// Mitsubishi GX Works2 project: Jesús Beato 2023-1283 #3   PLC: Q00J

PROGRAM MAIN
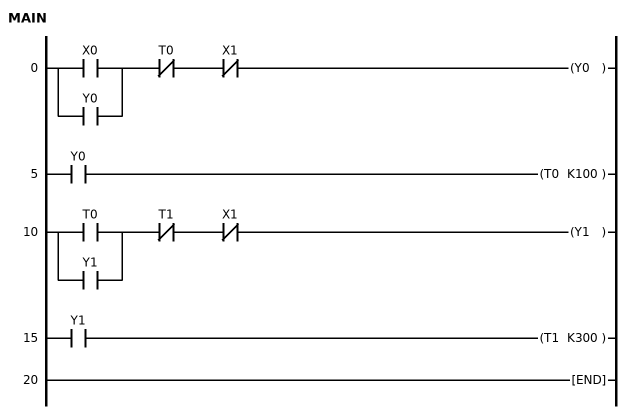
0     LD      X0
      OR      Y0
      ANI     T0
      ANI     X1
      OUT     Y0
5     LD      Y0
      OUT     T0 K100
10    LD      T0
      OR      Y1
      ANI     T1
      ANI     X1
      OUT     Y1
15    LD      Y1
      OUT     T1 K300
20    END
END_PROGRAM
